// TwinCAT 3 PLC project Untitled1
// ProgramVersion: 3.1.4024.0
// libraries:
//   Tc2_MC2, * (Beckhoff Automation GmbH)
//   Tc2_Standard, * (Beckhoff Automation GmbH)
//   Tc2_System, * (Beckhoff Automation GmbH)
//   Tc2_TcpIp, * (Beckhoff Automation GmbH)
//   Tc2_Utilities, * (Beckhoff Automation GmbH)
//   Tc3_Module, * (Beckhoff Automation GmbH)
// project tree:
//   GVLs/ GVL.TcGVL, GVL_HMI.TcGVL
//   / PlcTask.TcTTO
//   POUs/Alarm/ FB_Alarm.TcPOU
//   POUs/Main/ FB_Machine.TcPOU, MAIN.TcPOU
//   POUs/UniversalBlocks/Cylinder/ FB_Cylinder.TcPOU, FB_CylinderDiag.TcPOU, FB_CylinderTemp.TcPOU, FB_CylinderTempDiag.TcPOU, FB_CylinderTempRecord.TcPOU
//   POUs/UniversalBlocks/TCP IP/ FB_TCPServer.TcPOU
//   POUs/UniversalBlocks/Universal Digital Input/ FB_Input.TcPOU, I_Input.TcIO
//   POUs/UniversalBlocks/Universal Digital Output/ FB_Output.TcPOU, I_Output.TcIO
//   POUs/UniversalBlocks/Universal motor/ FB_Axis.TcPOU, FB_Axis_Multi_Master.TcPOU, FB_HomeableAxis.TcPOU, FB_HomeableEncAxis.TcPOU, I_UniversalMotor.TcIO
// real-time tasks:
//   TASK PlcTask: cycle T#10ms, priority 20, ADS port 350
// motion (NC):
//   TASK NC-Task 1 SAF: cycle T#2ms, priority 4, ADS port 501
//   TASK NC-Task 1 SVB: cycle T#10ms, priority 8, ADS port 511
//   AXIS Axis 1 (id 1)
// variable links:
//   Untitled1 Instance <-> NC-Task 1 SAF/Axes/Axis 1
//     PlcTask Inputs/MAIN.fbMachine.servo.AxisRef.NcToPlc <-> Outputs/ToPlc
//     PlcTask Outputs/MAIN.fbMachine.servo.AxisRef.PlcToNc <-> Inputs/FromPlc

CONFIGURATION Untitled1
    RESOURCE PLC ON TwinCAT3
        TASK PlcTask(INTERVAL := T#10ms, PRIORITY := 20);
        PROGRAM MAIN WITH PlcTask : MAIN;
    END_RESOURCE
END_CONFIGURATION

// ---- GVLs/GVL.TcGVL
{attribute 'qualified_only'}
VAR_GLOBAL		
		fbLocalTime	:	FB_LocalSystemTime;
		iYear		:	UINT;
		iMonth		:	UINT;
		iDay		:	UINT;
		iHour		:	UINT;
		iMinute		:	UINT;
		iSecond		:	UINT;
END_VAR

// ---- GVLs/GVL_HMI.TcGVL
{attribute 'qualified_only'}
VAR_GLOBAL
//Cylinder
//Input
	bMoveWorkCylinder1	: BOOL;
	bMoveBaseCylinder1	: BOOL;
	bMoveWorkCylinder2	: BOOL;
	bMoveBaseCylinder2	: BOOL;
	bMoveWorkCylinder3	: BOOL;
	bMoveBaseCylinder3	: BOOL;
	bMoveWorkCylinder4	: BOOL;
	bMoveBaseCylinder4	: BOOL;
//Cylinder
//Output
	bAtBasePosCylinder1	: BOOL;
	bAtWorkPosCylinder1	: BOOL;
	bAtBasePosCylinder2	: BOOL;
	bAtWorkPosCylinder2	: BOOL;
	bAtBasePosCylinder3	: BOOL;
	bAtWorkPosCylinder3	: BOOL;
	bAtBasePosCylinder4	: BOOL;
	bAtWorkPosCylinder4	: BOOL;

//Servo
//Input
	bMoveServo			: BOOL;
	rDistance			: LREAL;
	bStopServo			: BOOL;
	
//Servo
//Output
	rPosition			: LREAL;
	rVelocity			: LREAL;
	rEnable				: BOOL;
	bErrorServo			: BOOL;
//Tcp-ip server
//Input
	bConnect			: BOOL;
	bDisconnect			: BOOL;
	bSend				: BOOL;
	sDataSend			: STRING(255);
//Tcp-ip server
//Output
	bIsConnect			: BOOL;
	sLocalHost			: T_IPv4Addr;
	sLocalPort			: UDINT;
	sDataRev			: STRING(255);
	bErrorTcp			: BOOL;
//System
//Input
	bManual				: BOOL;
	bAuto				: BOOL;
	bStart				: BOOL;
	bReset				: BOOL;
	bStopSystem			: BOOL;
	bEStopSystem		: BOOL;
	
	bSensorCheck		: BOOL;
	bSensorOK			: BOOL;
	bSensorNG			: BOOL;
	
	bSensorBase1HMI		: BOOL;
	bSensorWork1HMI     : bool;
	bSensorBase2HMI     : bool;
	bSensorWork2HMI     : bool;
	bSensorBase3HMI     : bool;
	bSensorWork3HMI     : bool;
	bSensorBase4HMI     : bool;
	bSensorWork4HMI     : bool;
	
	bRunStep			: BOOL;
	bRun				: BOOL;
	
	bOnLightGreen		: BOOL;
	bOnLightYellow		: BOOL;
	bOnLightRed			: BOOL;
		
//System
//Output
	bIsReady			: BOOL;
	bLightGreen			: BOOL;
    bLightYellow	    : bool;
    bLightRed		    : bool;
                       
	iCounterOK			: INT;
	iCounterNG			: INT;
	bErrorSystem		: BOOL;
END_VAR

// ---- POUs/UniversalBlocks/Universal Digital Input/I_Input.TcIO
INTERFACE I_Input

PROPERTY Description : STRING
GET
END_GET
SET
END_SET
END_PROPERTY

PROPERTY Value : BOOL
GET
END_GET
END_PROPERTY

END_INTERFACE

// ---- POUs/UniversalBlocks/Universal Digital Output/I_Output.TcIO
INTERFACE I_Output

PROPERTY Description : STRING
GET
END_GET
SET
END_SET
END_PROPERTY

PROPERTY ManualMode : BOOL
GET
END_GET
SET
END_SET
END_PROPERTY

PROPERTY OutAuto : BOOL
GET
END_GET
SET
END_SET
END_PROPERTY

PROPERTY OutManual : BOOL
GET
END_GET
SET
END_SET
END_PROPERTY

END_INTERFACE

// ---- POUs/UniversalBlocks/Universal motor/I_UniversalMotor.TcIO
INTERFACE I_UniversalMotor

METHOD Abort : BOOL
VAR_INPUT
END_VAR
END_METHOD

PROPERTY ActualPosition : LREAL
GET
END_GET
END_PROPERTY

PROPERTY AxisReference : AXIS_REF
GET
END_GET
END_PROPERTY

METHOD Couple : BOOL
VAR_INPUT

END_VAR

VAR

END_VAR
END_METHOD

PROPERTY Coupleable : BOOL
GET
END_GET
SET
END_SET
END_PROPERTY

PROPERTY Coupled : BOOL
GET
END_GET
END_PROPERTY

METHOD Decouple : BOOL
VAR_INPUT
END_VAR
VAR
END_VAR
END_METHOD

METHOD Home : BOOL // Start axis homing
VAR_INPUT
END_VAR
END_METHOD

PROPERTY Homed : BOOL
GET
END_GET
END_PROPERTY

PROPERTY Homingable : BOOL
GET
END_GET
SET
END_SET
END_PROPERTY

METHOD Init : BOOL
VAR_INPUT
END_VAR
END_METHOD

PROPERTY Initialized : BOOL
GET
END_GET
END_PROPERTY

METHOD Jog : BOOL
VAR_INPUT
	Distance	:	LREAL;
END_VAR
END_METHOD

PROPERTY MotorName : STRING
GET
END_GET
SET
END_SET
END_PROPERTY

METHOD MoveAbsolute : BOOL // Do action 2 request, for instance: 'Pick and place unit' change tool (additional inputs needed)
VAR_INPUT
	Position : LREAL;
END_VAR
END_METHOD

METHOD Reset : BOOL
VAR_INPUT
END_VAR
END_METHOD

PROPERTY Unit : STRING
GET
END_GET
SET
END_SET
END_PROPERTY

END_INTERFACE

// ---- POUs/Main/MAIN.TcPOU
PROGRAM MAIN
VAR
	fbMachine	: FB_Machine;
	bTimeValid	: BOOL;

END_VAR

fbMachine();
CurrentTime();

METHOD CurrentTime : BOOL
VAR_INPUT
END_VAR
GVL.fbLocalTime(bEnable := TRUE);

IF GVL.fbLocalTime.bValid THEN
	bTimeValid := TRUE;
END_IF

IF bTimeValid THEN
	GVL.iYear 	:= WORD_TO_UINT(GVL.fbLocalTime.systemTime.wYear);
	GVL.iMonth 	:= WORD_TO_UINT(GVL.fbLocalTime.systemTime.wMonth);
	GVL.iDay 	:= WORD_TO_UINT(GVL.fbLocalTime.systemTime.wDay);
	GVL.iHour 	:= WORD_TO_UINT(GVL.fbLocalTime.systemTime.wHour);
	GVL.iMinute := WORD_TO_UINT(GVL.fbLocalTime.systemTime.wMinute);
	GVL.iSecond := WORD_TO_UINT(GVL.fbLocalTime.systemTime.wSecond);
END_IF
END_METHOD

END_PROGRAM

// ---- POUs/Main/FB_Machine.TcPOU
FUNCTION_BLOCK FB_Machine
VAR_INPUT
	bManual	: FB_Input;
	bAuto	: FB_Input;
END_VAR
VAR_OUTPUT
	bError		: BOOL;
	iErrorId	: INT;
END_VAR

VAR
	iStepGeneral	: INT;
	bISError		: BOOL;
	bIsReady		: BOOL;
	trig3s			: ton :=(pt:=T#3S);
	trig1s			: ton :=(pt:=T#1S);
	trig500ms		: ton :=(pt:=T#500MS);
	trigCylin1		: ton;
	tTimeCylin1		: TIME	:= T#0.5S;
	trigCylin2		: ton;
	tTimeCylin2		: TIME	:= T#2S;
	bLightGreen		: FB_Output;
	bLightYellow	: FB_Output;
	bLightRed		: FB_Output;
	bStart			: FB_Input;
	bReset			: FB_Input;
	bSensorCheck	: FB_Input;
	bSensorOK		: FB_Input;
	bSensorNG		: FB_Input;
	bStop			: FB_Input;
	bEStop			: FB_Input;
	bStopTem		: BOOL;
	bRunStep		: BOOL := FALSE;
	bRun			: BOOL := FALSE;
	trigStep		: r_trig;
	trigSensorOK	: r_trig;
	trigSensorNG	: r_trig;
	iCounterOK		: INT;
	iCounterNG		: INT;
	bOnLightGreen	: BOOL;
	bOnLightYellow	: BOOL;
	bOnLightRed		: BOOL;
	//Tcp-ip
	trigTCp			: r_trig;
	fbTcpServer		: FB_TCPServer;
	sLocalHost		: T_IPv4Addr := '';
	nLocalPort		: UDINT := 9000;
	sNetId			: T_AmsNetId := '';  //'5.30.162.44.1.1';
	sDataRev		: STRING(255);
	sDataSend		: STRING(255);
	bConnect		: BOOL;
	bDisconnect		: BOOL;
	bSend			: BOOL;
	//servo
	servo			: FB_Axis;
	bMoveServo		: BOOL;
	rDistance		: LREAL;
	bStopServo		: BOOL;
	//cylinder
	cylinder1		: FB_CylinderDiag;
	cylinder2		: FB_CylinderDiag;
	cylinder3		: FB_CylinderDiag;
	cylinder4		: FB_CylinderDiag;
	//Alarm
	servoAlarm		: FB_Alarm;
	tcpServerAlarm	: Fb_Alarm;
	cylinderAlarm	: FB_Alarm;
	
	bMoveWorkCylinder1	: BOOL;
	bMoveBaseCylinder1	: BOOL;
	bMoveWorkCylinder2	: BOOL;
	bMoveBaseCylinder2	: BOOL;
	bMoveWorkCylinder3	: BOOL;
	bMoveBaseCylinder3	: BOOL;
	bMoveWorkCylinder4	: BOOL;
	bMoveBaseCylinder4	: BOOL;
	
	bManualHMI		: BOOL;
	bAutoHMI		: BOOL;
	bStartHMI		: BOOL;
	bResetHMI		: bool;
	bStopHMI		: bool;
	bEStopHMI		: bool;
	bSensorCheckHMI	: bool;
	bSensorOKHMI	: bool;
	bSensorNGHMI	: BOOL;
	bSensorBase1HMI	: BOOL;
	bSensorWork1HMI	: BOOL;
	bSensorBase2HMI	: BOOL;
	bSensorWork2HMI	: BOOL;
	bSensorBase3HMI	: BOOL;
	bSensorWork3HMI	: BOOL;
	bSensorBase4HMI	: BOOL;
	bSensorWork4HMI	: BOOL;
	
	iStepRun: INT := 0;
	iStepAuto: INT := 0;
	bCheck : BOOL;
	bFirstCycle	: BOOL := TRUE;
END_VAR

StateMachine();
AssignHMI();
servo();
fbTcpServer();
//Menu mode
IF bManual.Value OR bManualHMI THEN
	iStepRun	:= 20;
END_IF
IF bAuto.Value OR bAutoHMI THEN
	iStepRun	:= 10;
END_IF
//Reset
IF bReset.Value OR bResetHMI THEN
	iStepGeneral := 0;
END_IF
//Stop
IF bStop.Value OR bStopHMI THEN
	bStopTem := TRUE;
END_IF
IF bEStop.Value OR bEStopHMI THEN
	iStepGeneral	:= 99;
END_IF
//Error
bError := servoAlarm.Get() OR tcpServerAlarm.Get() OR cylinderAlarm.Get();

METHOD AssignHMI : BOOL
VAR_INPUT
END_VAR
//Cylinder              
//Input                 
bMoveWorkCylinder1		:=	GVL_HMI.bMoveWorkCylinder1	;
bMoveBaseCylinder1		:=	GVL_HMI.bMoveBaseCylinder1	;
bMoveWorkCylinder2		:=	GVL_HMI.bMoveWorkCylinder2	;
bMoveBaseCylinder2		:=	GVL_HMI.bMoveBaseCylinder2	;
bMoveWorkCylinder3		:=	GVL_HMI.bMoveWorkCylinder3	;
bMoveBaseCylinder3		:=	GVL_HMI.bMoveBaseCylinder3	;
bMoveWorkCylinder4		:=	GVL_HMI.bMoveWorkCylinder4	;
bMoveBaseCylinder4		:=	GVL_HMI.bMoveBaseCylinder4	;

bSensorBase1HMI			:= GVL_HMI.bSensorBase1HMI;
bSensorWork1HMI         := GVL_HMI.bSensorWork1HMI;
bSensorBase2HMI         := GVL_HMI.bSensorBase2HMI;
bSensorWork2HMI         := GVL_HMI.bSensorWork2HMI;
bSensorBase3HMI         := GVL_HMI.bSensorBase3HMI;
bSensorWork3HMI         := GVL_HMI.bSensorWork3HMI;
bSensorBase4HMI         := GVL_HMI.bSensorBase4HMI;
bSensorWork4HMI         := GVL_HMI.bSensorWork4HMI;
//Cylinder                                          
//Output                
GVL_HMI.bAtBasePosCylinder1	:= cylinder1.bState_AtBasePos OR cylinder1.bState_MoveToBase;
GVL_HMI.bAtWorkPosCylinder1	:= cylinder1.bState_AtWorkPos OR cylinder1.bState_MoveToWork;
GVL_HMI.bAtBasePosCylinder2	:= cylinder2.bState_AtBasePos OR cylinder2.bState_MoveToBase;
GVL_HMI.bAtWorkPosCylinder2	:= cylinder2.bState_AtWorkPos OR cylinder2.bState_MoveToWork;
GVL_HMI.bAtBasePosCylinder3	:= cylinder3.bState_AtBasePos OR cylinder3.bState_MoveToBase;
GVL_HMI.bAtWorkPosCylinder3	:= cylinder3.bState_AtWorkPos OR cylinder3.bState_MoveToWork;
GVL_HMI.bAtBasePosCylinder4	:= cylinder4.bState_AtBasePos OR cylinder4.bState_MoveToBase;
GVL_HMI.bAtWorkPosCylinder4	:= cylinder4.bState_AtWorkPos OR cylinder4.bState_MoveToWork;
                        
//Servo                 
//Input                 
bMoveServo	:=	GVL_HMI.bMoveServo	;		
rDistance	:=	GVL_HMI.rDistance	;		
bStopServo	:=	GVL_HMI.bStopServo	;		
	                    
//Servo                 
//Output                
GVL_HMI.rPosition	:= servo.ActualPosition;		
GVL_HMI.rVelocity	:= servo.ActualVelocity;
GVL_HMI.rEnable		:= servo.Enabled;	
gvl_hmi.bErrorServo	:= servo.AnyError;
//Tcp-ip server         
//Input                 
bConnect	:= GVL_HMI.bConnect		;	
bDisconnect	:= GVL_HMI.bDisconnect	;		
bSend		:= GVL_HMI.bSend		;		
sDataSend	:= GVL_HMI.sDataSend	;
fbTcpServer.LocalHost	:=GVL_HMI.sLocalHost;
fbTcpServer.LocalPort	:=GVL_HMI.sLocalPort;		
//Tcp-ip server         
//Output                
GVL_HMI.bIsConnect	:= fbTcpServer.IsConnect;		
GVL_HMI.sDataRev	:= fbTcpServer.DataRev;
GVL_HMI.bErrorTcp	:= fbTcpServer.Error;
//System                
//Input                 
bRunStep			:= gvl_hmi.bRunStep;
bRun	            := gvl_hmi.bRun;
bManualHMI			:= GVL_HMI.bManual		;		
bAutoHMI			:= GVL_HMI.bAuto		;		
bStartHMI			:= GVL_HMI.bStart		;		
bResetHMI			:= GVL_HMI.bReset		;		
bStopHMI			:= GVL_HMI.bStopSystem	;		 	
bEStopHMI			:= GVL_HMI.bEStopSystem	;		                 
bSensorCheckHMI		:= GVL_HMI.bSensorCheck	;		
bSensorOKHMI		:= GVL_HMI.bSensorOK	;		
bSensorNGHMI		:= GVL_HMI.bSensorNG	;
bOnLightGreen			:= gvl_hmi.bOnLightGreen;
bOnLightYellow		:= gvl_hmi.bOnLightGreen;
bOnLightRed		  	:= gvl_hmi.bOnLightGreen;
		                
//System                
//Output

gvl_hmi.bIsReady		:= bIsReady;               
GVL_HMI.iCounterOK		:= iCounterOK;	
GVL_HMI.iCounterNG		:= iCounterOK;		
GVL_HMI.bErrorSystem	:= bError;

GVL_HMI.bLightGreen		:= 	bLightGreen.OutAuto;
GVL_HMI.bLightYellow    :=  bLightYellow.OutAuto;
GVL_HMI.bLightRed	    :=  bLightRed.OutAuto;
END_METHOD

METHOD PRIVATE StateAuto : BOOL
VAR

END_VAR

CASE iStepAuto OF
	0: //run servo 10
			trigStep(clk:=bRun);
			IF NOT bRunStep OR trigStep.Q THEN
				iStepAuto := iStepAuto + 1;
			END_IF
	1:
		IF NOT servo.AnyError AND servo.Enabled THEN
			IF servo.ActualPosition <> 10 THEN
				servo.MoveAbsolute(Position := 10);
			END_IF
		ELSE
			iStepAuto := 99;
		END_IF
		IF servo.ActualPosition = 10 THEN
			trigStep(clk:=bRun);
			IF NOT bRunStep OR trigStep.Q THEN
				iStepAuto := iStepAuto + 1;
			END_IF
		END_IF

	2: // run cylinder 1
		IF bSensorCheck.Value OR bSensorCheckHMI THEN
			bCheck := TRUE;
		END_IF		
		
		IF bCheck THEN
			IF NOT cylinder1.bError THEN
				cylinder1.MoveToWork();
			ELSE
				iStepAuto	:= 99;
			END_IF
			trigCylin1(in:= cylinder1.bState_AtWorkPos OR bSensorWork1HMI,pt:=tTimeCylin1);
			IF trigCylin1.Q THEN
				cylinder1.MoveToBase();
				bCheck	:= FALSE;
			END_IF
		END_IF
			
			
		IF cylinder1.bState_AtBasePos OR bSensorBase1HMI AND( NOT bSensorCheck.Value OR NOT bSensorCheckHMI )THEN
			trigStep(clk:=bRun);
			IF NOT bRunStep OR trigStep.Q THEN
				iStepAuto := iStepAuto + 1;
			END_IF
		END_IF
	3:// run servo 70
		IF NOT servo.AnyError THEN
			IF servo.ActualPosition <> 70 THEN
				servo.MoveAbsolute(Position := 70);
			END_IF			
		ELSE
			iStepAuto := 99;
		END_IF
		IF servo.ActualPosition = 70 THEN
			bCheck	:= TRUE;
			trigStep(clk:=bRun);
			IF NOT bRunStep OR trigStep.Q THEN
				iStepAuto := iStepAuto + 1;
			END_IF
		END_IF
		
	4://run cylin 2
		IF bCheck THEN
			IF NOT cylinder2.bError THEN
				cylinder2.MoveToWork();
			ELSE
				iStepAuto	:= 99;
			END_IF
			trigCylin2(in:= cylinder2.bState_AtWorkPos OR bSensorWork2HMI,pt:=tTimeCylin2);
			IF trigCylin2.Q THEN
				cylinder2.MoveToBase();
				bCheck	:= FALSE;
			END_IF
		END_IF
		IF NOT bCheck THEN
			trigStep(clk:=bRun);
			IF NOT bRunStep OR trigStep.Q THEN
				iStepAuto := iStepAuto + 1;
			END_IF
		END_IF

	5://run servo 130
		IF NOT servo.AnyError THEN
			IF servo.ActualPosition <> 130 THEN
				servo.MoveAbsolute(Position := 130);
			END_IF
		ELSE
			iStepAuto := 99;
		END_IF
		
		IF servo.ActualPosition = 130 THEN
			bCheck	:= TRUE;
			trigStep(clk:=bRun);
			IF NOT bRunStep OR trigStep.Q THEN
				iStepAuto := iStepAuto + 1;
			END_IF
		END_IF
	6:// trigger camera
		IF bCheck THEN
			IF fbTcpServer.IsConnect THEN
				fbTcpServer.SendData(DataSend :='CHE,1');
				bCheck := FALSE;
			ELSE
				iStepAuto := 99;
			END_IF
		END_IF
	
		IF NOT bCheck THEN
			trigStep(clk:=bRun);
			IF NOT bRunStep OR trigStep.Q THEN
				iStepAuto := iStepAuto + 1;
			END_IF
		END_IF
	
	7:// check camera
		sDataRev := fbTcpServer.DataRev;
		trigStep(clk:=bRun);
		IF NOT bRunStep OR trigStep.Q THEN
			IF sDataRev = 'CAM,1,OK' THEN
					iStepAuto := iStepAuto + 1;
			END_IF
			IF sDataRev = 'CAM,1,NG' THEN
					iStepAuto := iStepAuto + 2;
			END_IF
		END_IF
		
	8:// run servo 190
		IF NOT servo.AnyError THEN
			IF servo.ActualPosition <> 190 THEN
				servo.MoveAbsolute(Position := 190);
			END_IF
		ELSE
			iStepAuto := 99;
		END_IF
		
		IF servo.ActualPosition = 190 THEN
			bCheck	:= TRUE;
			trigStep(clk:=bRun);
			IF NOT bRunStep OR trigStep.Q THEN
				iStepAuto := iStepAuto + 2;
			END_IF
		END_IF

	9:// run servo 210
		IF NOT servo.AnyError THEN
			IF servo.ActualPosition <> 210 THEN
				servo.MoveAbsolute(Position := 210);
			END_IF
		ELSE
			iStepAuto := 99;
		END_IF
		IF servo.ActualPosition = 210 THEN
			bCheck	:= TRUE;
			trigStep(clk:=bRun);
			IF NOT bRunStep OR trigStep.Q THEN
				iStepAuto := iStepAuto + 2;
			END_IF
		END_IF
	10://run cylin 3
		IF bCheck THEN
			IF NOT cylinder3.bError THEN
				cylinder3.MoveToWork();
				IF cylinder3.bState_AtWorkPos OR bSensorWork3HMI THEN
					cylinder3.MoveToBase();
					bCheck := FALSE;
				END_IF
			ELSE
				iStepAuto	:= 99;
			END_IF
		END_IF
		
		IF NOT bCheck THEN
			trigStep(clk:=bRun);
			IF NOT bRunStep OR trigStep.Q THEN
				iStepAuto := iStepAuto + 2;
			END_IF
		END_IF

	11://run cylin 4
		IF bCheck THEN
			IF NOT cylinder4.bError THEN
				cylinder4.MoveToWork();
				IF cylinder4.bState_AtWorkPos OR bSensorWork4HMI THEN
					cylinder4.MoveToBase();
					bCheck := FALSE;
				END_IF
			ELSE
				iStepAuto	:= 99;
			END_IF
		END_IF
		
		IF NOT bCheck THEN
			trigStep(clk:=bRun);
			IF NOT bRunStep OR trigStep.Q THEN
				iStepAuto := iStepAuto + 1;
			END_IF
		END_IF

	12:// counter
		trigSensorOK(clk:=bSensorOK.Value OR bSensorOKHMI);
		trigSensorNG(clk:=bSensorNG.Value OR bSensorNGHMI);
		IF trigSensorOK.Q THEN
			icounterOK := icounterOK + 1;
		END_IF
		IF trigSensorNG.Q THEN
			icounterNG := icounterNG + 1;
		END_IF
		IF NOT bStopTem THEN
			iStepAuto := 0;
		END_IF
	99://Error
		iStepGeneral := 99;
		
		
END_CASE
END_METHOD

METHOD PRIVATE StateError : BOOL
VAR
	bfirstCycle	: bool := true;
END_VAR
IF bfirstCycle THEN
	bfirstCycle:= FALSE;
	IF servo.AnyError THEN
		servoAlarm.Set(bIn := TRUE);
		servoAlarm.Description := 'Servo bi loi';
	END_IF
	IF fbTcpServer.Error THEN
		tcpServerAlarm.Set(bIn := TRUE);
		tcpServerAlarm.Description := 'TCP-IP Server bi loi';
		END_IF
	IF NOT fbTcpServer.IsConnect THEN
		tcpServerAlarm.Set(bIn := TRUE);
		tcpServerAlarm.Description := 'Khong co Client nao ket noi';
	END_IF
END_IF
	

trig1s(IN := TRUE);
IF trig1s.Q THEN
	trig1s(IN := TRUE);
	bLightRed.OutAuto := NOT bLightRed.OutAuto;
END_IF

IF bReset.Value THEN
	iStepGeneral := 0;
END_IF
END_METHOD

METHOD PRIVATE StateInit : BOOL
VAR
	
END_VAR
//init cylin
cylinder1.MoveToBase();
cylinder1.Reset();
cylinder2.MoveToBase();
cylinder2.Reset();
cylinder3.MoveToBase();
cylinder3.Reset();
cylinder4.MoveToBase();
cylinder4.Reset();
//init servo
servo.Reset();
servo.Override := 100;
servo.Init();
servo.MoveAbsolute(Position:=0);
//Init tcp-ip
IF NOT fbTcpServer.IsConnect THEN
	IF bFirstCycle THEN
		bFirstCycle := FALSE;
		fbTcpServer.Disconnect();
		fbTcpServer.LocalHost	:= sLocalHost;
		fbTcpServer.LocalPort	:= nLocalPort;
		fbTcpServer.NetId		:= sNetId;
		fbTcpServer.Connect();
	END_IF
END_IF

bLightGreen.OutAuto 	:= FALSE;
bLightYellow.OutAuto 	:= FALSE;
blightRed.OutAuto 		:= FALSE;

bCheck					:= FALSE;
iStepAuto				:= 0;
IF servo.ActualPosition = 0 THEN
	iStepGeneral			:= iStepGeneral + 1;
END_IF
END_METHOD

METHOD private StateMachine : BOOL
VAR_INPUT
END_VAR
CASE iStepGeneral OF
	0: 
		StateInit();
	1:
		StateUninitialized();
	2:
		StateReady();
	10:
		StateRun();
	20:
		StateRunDone();
	30:
		StateStop();
	40:
		StateStopDone();
	99:
		StateError();
	
END_CASE
END_METHOD

METHOD PRIVATE StateManual : BOOL
VAR_INPUT
END_VAR
//cylinder
IF bMoveWorkCylinder1 THEN
	cylinder1.MoveToWork();
	bMoveWorkCylinder1 := FALSE;
END_IF
IF bMoveBaseCylinder1 THEN
	cylinder1.MoveToBase();
	bMoveBaseCylinder1 := FALSE;
END_IF
IF bMoveWorkCylinder2 THEN
	cylinder2.MoveToWork();
	bMoveWorkCylinder2 := FALSE;
END_IF
IF bMoveBaseCylinder2 THEN
	cylinder2.MoveToBase();
	bMoveBaseCylinder2 := FALSE;
END_IF
IF bMoveWorkCylinder3 THEN
	cylinder3.MoveToWork();
	bMoveWorkCylinder3 := FALSE;
END_IF
IF bMoveBaseCylinder3 THEN
	cylinder3.MoveToBase();
	bMoveBaseCylinder3 := FALSE;
END_IF
IF bMoveWorkCylinder4 THEN
	cylinder4.MoveToWork();
	bMoveWorkCylinder4 := FALSE;
END_IF
IF bMoveBaseCylinder4 THEN
	cylinder4.MoveToBase();
	bMoveBaseCylinder4 := FALSE;
END_IF
//servo
IF bMoveServo THEN
	servo.Jog(Distance:=rDistance);
	bMoveServo := FALSE;
END_IF
IF bStopServo THEN
	bStopServo := FALSE;
	servo.Stop();
END_IF
//TCP-Ip
IF bConnect THEN
	fbTcpServer.Connect();
	bConnect := FALSE;
END_IF
IF bDisconnect THEN
	fbTcpServer.Disconnect();
	bDisconnect := FALSE;
END_IF
IF bSend THEN
	fbTcpServer.SendData(DataSend := sDataSend);
	bSend := FALSE;
END_IF
//system
bLightGreen.OutAuto		:= bOnLightGreen	;
bLightYellow.OutAuto    := bOnLightYellow	;
bLightRed.OutAuto       := bOnLightRed		;
END_METHOD

METHOD PRIVATE StateReady : BOOL
VAR_INPUT
END_VAR
trig500ms(in := TRUE);
IF bIsReady AND trig500ms.Q THEN
	trig500ms(in := FALSE);
	bLightGreen.OutAuto := NOT bLightGreen.OutAuto;
END_IF

IF bStart.Value OR bStartHMI THEN
	iStepGeneral := 10;
END_IF
END_METHOD

METHOD PRIVATE StateRun : BOOL
VAR_INPUT
END_VAR
CASE iStepRun OF
	10:
		StateAuto();
		bLightGreen.OutAuto := TRUE;
	20:
		StateManual();
END_CASE
END_METHOD

METHOD PRIVATE StateRunDone : BOOL
VAR_INPUT
END_VAR
END_METHOD

METHOD PRIVATE StateStop : BOOL
VAR_INPUT
END_VAR
END_METHOD

METHOD PRIVATE StateStopDone : BOOL
VAR_INPUT
END_VAR
END_METHOD

METHOD PRIVATE StateUninitialized : BOOL
VAR_INPUT
END_VAR
bISError := servo.AnyError OR fbTcpServer.Error OR fbTcpServer.Error ;
//bIsReady := cylinder1.bState_AtBasePos AND cylinder2.bState_AtBasePos AND cylinder3.bState_AtBasePos AND cylinder4.bState_AtBasePos AND fbTcpServer.IsConnect AND servo.Enabled;
bIsReady := TRUE;
		
IF bIsError THEN
	iStepGeneral := 99;
END_IF

IF NOT bIsReady THEN
	bLightYellow.OutAuto := TRUE;
END_IF

IF bIsReady THEN
	iStepGeneral := 2;
END_IF
IF NOT bIsReady THEN
	IF bReset.Value OR bResetHMI THEN
		iStepGeneral := 0;
	END_IF
END_IF
END_METHOD

END_FUNCTION_BLOCK

// ---- POUs/UniversalBlocks/Universal Digital Input/FB_Input.TcPOU
FUNCTION_BLOCK FB_Input IMPLEMENTS I_Input
VAR_INPUT
END_VAR
VAR_OUTPUT
END_VAR
VAR
	sDescription			:	STRING; //Description of the physical input
	bIn				AT %I*	:	BOOL;	// Physical input
	bRisingTrigger			:	BOOL;
	bFallingTrigger			:	BOOL;
	rtIn					:	R_TRIG; //Rising edge of the input
	ftIn					:	F_TRIG; //Falling edge of the input	
END_VAR

PROPERTY Description : STRING
GET
Description := sDescription;
END_GET
SET
sDescription := Description;
END_SET
END_PROPERTY

PROPERTY Value : BOOL
GET
Value := bIn;
END_GET
END_PROPERTY

END_FUNCTION_BLOCK

// ---- POUs/UniversalBlocks/Universal Digital Output/FB_Output.TcPOU
// Function block used for physical output control
FUNCTION_BLOCK FB_Output IMPLEMENTS I_Output
VAR_INPUT

END_VAR
VAR_OUTPUT

END_VAR
VAR
	bOut	AT %Q*	:	BOOL;	// Physical output
	sDescription	:	STRING;	// Description of the output
	bOutAuto		:	BOOL;	// This value will be used in automatic mode
	bManualMode		:	BOOL;	// Turns on and off manual mode
	bOutManual		:	BOOL;	// This value will be used in manual mode
END_VAR

{attribute 'monitoring' := 'variable'}
PROPERTY Description : STRING
GET
Description := sDescription;
END_GET
SET
sDescription := Description;
END_SET
END_PROPERTY

{attribute 'monitoring' := 'variable'}
PROPERTY ManualMode : BOOL
GET
ManualMode := bManualMode;
END_GET
SET
bManualMode := ManualMode;
END_SET
END_PROPERTY

{attribute 'monitoring' := 'variable'}
PROPERTY OutAuto : BOOL
GET
OutAuto := bOut;
END_GET
SET
bOutAuto := OutAuto;
IF NOT bManualMode THEN
	bOut := bOutAuto;
END_IF
END_SET
END_PROPERTY

{attribute 'monitoring' := 'variable'}
PROPERTY OutManual : BOOL
GET
OutManual := bOut;
END_GET
SET
bOutManual := OutManual;
IF bManualMode THEN
	bOut := bOutManual;
END_IF
END_SET
END_PROPERTY

END_FUNCTION_BLOCK

// ---- POUs/UniversalBlocks/TCP IP/FB_TCPServer.TcPOU
FUNCTION_BLOCK FB_TCPServer

VAR
	sLocalHost: T_IPv4Addr;
	nLocalPort: UDINT := 9000;
	//bStartCommunication : BOOL;
	sNetId	:T_AmsNetId;
	//bSent	: BOOL;

	bConnected: BOOL;
	sSendData: STRING(255);
	bBusy: BOOL;	
	bError: BOOL;
	nErrorID: UDINT;
	sDataRev: STRING(255);

	//iState: INT;
	hListener: T_HSOCKET;
	hSocket: T_HSOCKET;
	fbSocketAccept: FB_SocketAccept;
	fbSocketListen: FB_SocketListen;
	fbSocketReceive: FB_SocketReceive;
	fbSocketClose: FB_SocketClose;
	fbSocketCloseAll: FB_SocketCloseAll;
	fbSocketSend: FB_SocketSend;
	bAcceptExecute: BOOL;
	sReadData: STRING(255);
	ReceiveCounter: UDINT;
	bSocketCloseError: BOOL;
	nSocketCloseError: UDINT;
	//bSendTrigger: BOOL;
	//sData : STRING(255);
	iStepGeneral	: INT := 0;
	iStepStop		: INT := 0;
END_VAR

StateMachine();
IF bError THEN
	iStepGeneral := 50;
END_IF

METHOD Connect : BOOL
VAR_INPUT
END_VAR
IF NOT bConnected AND NOT bError THEN
	iStepGeneral := 1;
END_IF
END_METHOD

PROPERTY DataRev : String(255)
GET
DataRev := sDataRev;
END_GET
END_PROPERTY

METHOD Disconnect : BOOL
VAR_INPUT
END_VAR
iStepGeneral := 50;
END_METHOD

PROPERTY Error : bool
GET
Error	:= bError;
END_GET
END_PROPERTY

PROPERTY IsConnect : bool
GET
IsConnect	:= bConnected;
END_GET
END_PROPERTY

PROPERTY LocalHost : T_IPv4Addr
SET
sLocalHost	:= LocalHost;
END_SET
END_PROPERTY

PROPERTY LocalPort : UDINT
SET
//nLocalPort	:= LocalPort;
END_SET
END_PROPERTY

PROPERTY NetId : T_AmsNetId
SET
sNetId	:= NetId;
END_SET
END_PROPERTY

METHOD SendData : BOOL
VAR_INPUT
	DataSend	: STRING(255);
END_VAR
sSendData := DataSend;
IF bConnected OR bError THEN
	IF iStepGeneral = 30 THEN
		iStepGeneral := 40;
	END_IF
END_IF
END_METHOD

METHOD private StateAccept : BOOL
VAR_INPUT
END_VAR
fbSocketAccept(																
		sSrvNetId:= sNetId, 		
		hListener:= hListener, 													
		bExecute:= TRUE, 
		tTimeout:= T#4S, 
		bAccepted=> , 
		bBusy=> bBusy, 
		bError=> bError, 
		nErrId=> nErrorID,
		hSocket=> hSocket);														
	IF NOT fbSocketAccept.bBusy THEN
		fbSocketAccept(bExecute:= FALSE);
	END_IF

	IF bError THEN
		iStepGeneral := 50; 
	ELSIF hSocket.handle <> 0 THEN
		iStepGeneral := iStepGeneral + 10; 
		bConnected := TRUE;
	END_IF
END_METHOD

METHOD PRIVATE StateClose : BOOL
VAR_INPUT
END_VAR
CASE iStepStop OF
0:	// Error Handling	
	fbSocketClose(																// Close Listener-Socket
		sSrvNetId:= sNetId, 
		hSocket:= hListener, 
		bExecute:= TRUE, 
		tTimeout:= T#4S, 
		bBusy=> , 
		bError=> bError, 
		nErrId=> nErrorID);		
	IF (NOT fbSocketClose.bBusy) OR fbSocketClose.bError THEN
		hListener.handle := 0;
		iStepStop := iStepStop + 1;
	END_IF
1:	
	fbSocketClose(bExecute := FALSE);
	iStepStop := iStepStop + 1;
2:
	fbSocketClose(																// Close Connection Socket
		sSrvNetId:= sNetId, 
		hSocket:= hSocket, 
		bExecute:= TRUE, 
		tTimeout:= T#4S, 
		bBusy=> , 
		bError=> bError, 
		nErrId=> nErrorID);
	IF NOT (fbSocketClose.bBusy) OR fbSocketClose.bError THEN
		hSocket.handle 	:= 0;	
		iStepGeneral 	:= 0;
		iStepStop		:= 0;
		bConnected 		:= FALSE;
	END_IF
END_CASE
END_METHOD

METHOD PRIVATE StateInit : BOOL
VAR_INPUT
END_VAR
fbSocketCloseAll(
		sSrvNetId:= sNetId, 
		bExecute:= TRUE, 
		tTimeout:= T#3S, 
		bBusy=> , 
		bError=> bSocketCloseError, 
		nErrId=> nSocketCloseError);

IF NOT (fbSocketCloseAll.bBusy OR fbSocketCloseAll.bError) THEN
		fbSocketCloseAll(bExecute:= FALSE);
		fbSocketListen(bExecute := FALSE);
		fbSocketAccept(bExecute := FALSE);
		fbSocketClose(bExecute:= FALSE);
		bConnected	:= FALSE;
		bBusy 		:= TRUE;
		iStepGeneral := 10;
END_IF
END_METHOD

METHOD PRIVATE StateListen : BOOL
VAR_INPUT
END_VAR
fbSocketListen(																
		sSrvNetId:= sNetId, 														
		sLocalHost:= sLocalHost, 												
		nLocalPort:= nLocalPort, 												
		bExecute:= TRUE, 
		tTimeout:= T#4S, 
		bBusy=> bBusy, 
		bError=> bError, 
		nErrId=> nErrorID,
		hListener=> hListener);													
		
	IF hListener.handle <> 0 THEN
		iStepGeneral := iStepGeneral + 10;	
	ELSIF bError THEN
		iStepGeneral := 50;
	END_IF
END_METHOD

METHOD PRIVATE StateMachine : BOOL
VAR_INPUT
END_VAR
CASE iStepGeneral OF
	1:
		StateInit();
	10:
		StateListen();
	20:
		StateAccept();
	30:
		StateReceive();
	40:
		StateSend();
	50:
		StateClose();
END_CASE
END_METHOD

METHOD PRIVATE StateReceive : BOOL
VAR_INPUT
END_VAR
fbSocketReceive(															
		sSrvNetId:= sNetId, 
		hSocket:= hSocket, 
		cbLen:= SIZEOF(sReadData) , 
		pDest:= ADR(sReadData), 
		bExecute:= TRUE, 														
		tTimeout:= T#4S, 
		bBusy=> , 
		bError=> bError, 
		nErrId=> nErrorID,
		nRecBytes=> );
		
	IF NOT fbSocketReceive.bBusy THEN
		fbSocketReceive(bExecute := FALSE);
		IF fbSocketReceive.nRecBytes <> 0 THEN									
			sDataRev := sReadData;
		END_IF
	END_IF
	
	IF fbSocketReceive.bError OR(NOT bConnected) THEN					
		iStepGeneral := 50;
	END_IF
END_METHOD

METHOD PRIVATE StateSend : BOOL
VAR_INPUT
END_VAR
fbSocketSend(																// Send Data to client
		sSrvNetId:= sNetId, 
		hSocket:= hSocket, 
		cbLen:= SIZEOF(sSendData), 
		pSrc:= ADR(sSendData),
		bExecute:= TRUE, 
		tTimeout:= T#3S, 
		bBusy=> , 
		bError=> bError, 
		nErrId=> nErrorID);	
	
	IF NOT fbSocketSend.bBusy THEN												// Switch back to receiving state after sending
		iStepGeneral := iStepGeneral - 10;
	ELSIF fbSocketSend.bError OR NOT bConnected THEN
		iStepGeneral := 50;													// Close connection in case of error 
	END_IF
END_METHOD

END_FUNCTION_BLOCK

// ---- POUs/UniversalBlocks/Universal motor/FB_Axis.TcPOU
FUNCTION_BLOCK FB_Axis IMPLEMENTS I_UniversalMotor
VAR_OUTPUT

END_VAR
VAR	
		// =============== Axis reference =========================
	AxisRef			: AXIS_REF;				// Axis reference (process data plc/nc)
	
	//Motors data
	sMotorName	:	STRING := 'Motor';
	sUnits		:	STRING := 'mm';


	iNumberOfInstance	: SINT := 1; //numebr of currently used instance of MC_MoveVelocity
	// =============== Done signals of Halt and Reset =========
	bResetDone		: BOOL;					// Status of function block MC_Reset
	bHaltDone		: BOOL;					// Status of function block MC_Halt

	// =============== State variables ========================
	bStatusEnable	: BOOL;					// Enable feedback
	
	// =============== Motion parameters, override =====================
	lrVelocityAuto			: LREAL := 2;			// Target velocity
	lrAccelerationAuto		: LREAL := 100;			// Target acceleration
	lrDecelerationAuto		: LREAL := 100;			// Target deceleration
	lrJerkAuto				: LREAL := 100;			// Target jerk
	lrVelocityManual		: LREAL := 2;			// Target velocity
	lrAccelerationManual	: LREAL := 100;			// Target acceleration
	lrDecelerationManual	: LREAL := 100;			// Target deceleration
	lrJerkManual			: LREAL := 100;			// Target jerk
	lrOverride 				: LREAL := 100.0;		// Override 100%
	lrPosition				: LREAL := 0;			// Target Position
	mcBufferMode			: MC_BufferMode := MC_Aborting;		// buffer mode standard value
	lrDistanceToGo			: LREAL := 0; 			// distance do go for relative movement
	lrActualPosition		: LREAL; // actual postion
	
	// =============== Trigger function blocks ================
	fbTriggerHalt	: R_TRIG;				// Trigger to recognize rising edge of halt input
	fbTriggerReset	: R_TRIG;				// Trigger to recognize rising edge of reset input
	
//	// =============== Axis reference =========================
//	AxisRef			: AXIS_REF;				// Axis reference (process data plc/nc)
	
	// =============== Motion function blocks =================
	fbMcPower 		: MC_Power;				// FB for enable and override
	fbMcReset 		: MC_Reset;				// FB to reset axis
	fbMcStop 		: MC_Stop;				// FB to stop axis
	fbMcHalt		: MC_Halt;				// FB to halt axis

	fbMcMoveVelocity		: MC_MoveVelocity;		// FB to move axis (velocity movement)
	fbMcMoveAbsolute		: MC_MoveAbsolute;		// FB to move axis (absolute PTP movement)
	fbMcMoveRelative		: MC_MoveRelative;		// FB to move axis (relative PTP movement)
	fbReadActualVelocity	: MC_ReadActualVelocity; //FB to read actual velocity of axis
	fbReadActualPosition	: MC_ReadActualPosition;//FB to read actual position of axis
	
	bFirstCycle		:	BOOL := TRUE; // indicates first cycle
	iStepInit		:	INT; // step of initialization
	

	bMoveVelocity	:	BOOL; //do action 2 variable
	bMoveAbsolute	:	BOOL; //do action 3 variable
	bMoveRelative	:	BOOL; //do action 4 variable
	bStop			:	BOOL; //do action 5 variable

	iStepGeneral	:	INT; // step of main state of unit
	iStepAborting	:	INT;

	
	bManualMode		:	BOOL;
	
	
	fbAxisError		:	FB_Alarm;
	
	bCoupleable		:	BOOL;
	bHomingable		:	BOOL;
	bInitialized	:	BOOL;

	// =============== Error variables ========================
	bError			: BOOL;					// Error signal
	iErrorID		: UDINT;				// Error ID
	
END_VAR

IF bFirstCycle THEN
	bFirstCycle := FALSE;
END_IF
// cyclic
		StateMachine();
		
	// reset commands
		bMoveVelocity := FALSE;
		bMoveAbsolute := FALSE;
		bMoveRelative := FALSE;
		bStop := FALSE;
		
	// read error
		IF AxisRef.Status.Error THEN
			bError := TRUE;
			iErrorID :=  AxisRef.Status.ErrorID;
		END_IF
		
	// read pos
		fbReadActualPosition(Enable := TRUE, Axis:=AxisRef);
		lrActualPosition :=	fbReadActualPosition.Position;

	// error	
		//fbAxisError.Description := FUN_MergeStrings5(sMotorName, ' axis error number: ', UDINT_TO_STRING(iErrorID), '', '');
		//fbAxisError.Set(bError);

	// status bits
		bInitialized := iStepGeneral > 10;

METHOD Abort : BOOL // Abort axis, it will disable the power
VAR_INPUT
END_VAR
IF iStepGeneral <> 0 THEN
	iStepGeneral := -10;
END_IF
iStepInit := 0;

//Method output
	Abort := (iStepGeneral = 0);
END_METHOD

{attribute 'monitoring' := 'variable'}
PROPERTY AccelerationAuto : LREAL
GET
AccelerationAuto := lrAccelerationAuto;
END_GET
SET
lrAccelerationAuto := AccelerationAuto;
END_SET
END_PROPERTY

{attribute 'monitoring' := 'variable'}
PROPERTY AccelerationManual : LREAL
GET
AccelerationManual := lrAccelerationManual;
END_GET
SET
lrAccelerationManual := AccelerationManual;
END_SET
END_PROPERTY

{attribute 'monitoring' := 'variable'}
PROPERTY ActualPosition : LREAL
GET
ActualPosition := lrActualPosition;
END_GET
END_PROPERTY

{attribute 'monitoring' := 'variable'}
PROPERTY ActualVelocity : LREAL
GET
fbReadActualVelocity(Enable:=TRUE,Axis:=AxisRef);
ActualVelocity:=fbReadActualVelocity.ActualVelocity;
END_GET
END_PROPERTY

{attribute 'monitoring' := 'variable'}
PROPERTY AnyError : BOOL
GET
AnyError := bError;
END_GET
END_PROPERTY

PROPERTY AxisReference : AXIS_REF
GET
AxisReference := AxisRef;
END_GET
END_PROPERTY

{attribute 'monitoring' := 'variable'}
PROPERTY Buffering : BOOL // TRUE for Enable, FALSE for disable
SET
IF Buffering THEN
	mcBufferMode := MC_BlendingNext;
ELSE
	mcBufferMode := MC_Aborting;
END_IF;
END_SET
END_PROPERTY

METHOD Couple : BOOL
VAR_INPUT
END_VAR
VAR
END_VAR
END_METHOD

{attribute 'monitoring' := 'variable'}
PROPERTY Coupleable : BOOL
GET
Coupleable := bCoupleable;
END_GET
SET
bCoupleable := Coupleable;
END_SET
END_PROPERTY

{attribute 'monitoring' := 'variable'}
PROPERTY Coupled : BOOL
GET
Coupled := AxisRef.Status.Coupled;
END_GET
END_PROPERTY

{attribute 'monitoring' := 'variable'}
PROPERTY DecelerationAuto : LREAL
GET
DecelerationAuto := lrDecelerationAuto;
END_GET
SET
lrDecelerationAuto := DecelerationAuto;
END_SET
END_PROPERTY

{attribute 'monitoring' := 'variable'}
PROPERTY DecelerationManual : LREAL
GET
DecelerationManual := lrDecelerationManual;
END_GET
SET
lrDecelerationManual := DecelerationManual;
END_SET
END_PROPERTY

METHOD Decouple : BOOL
VAR_INPUT
END_VAR
VAR
END_VAR
END_METHOD

METHOD PROTECTED Enable
VAR_INPUT
	bEnable		: BOOL;
END_VAR
// =========================================================

fbMCPower(	Enable 			:= bEnable, 
			Enable_Positive	:= bEnable, 
			Enable_Negative	:= bEnable, 
			Override		:= lrOverride,
			Axis			:= AxisRef,
			Status			=> bStatusEnable);
			
IF fbMcPower.Error THEN
	bError		:= TRUE;
	iErrorID 	:= fbMcPower.ErrorID;
END_IF

AxisRef.ReadStatus();
//bMoves := AxisRef.Status.Moving;

// =========================================================
END_METHOD

{attribute 'monitoring' := 'variable'}
PROPERTY Enabled : BOOL
GET
Enabled := bStatusEnable;
END_GET
END_PROPERTY

METHOD FirstCycle : BOOL
VAR_INPUT
	//ipAlarmController	:	I_AlarmController;
	//ipHMIController		:	I_HMIController;
	sName				:	STRING;
END_VAR
THIS^.sMotorName := sName;

//THIS^.ipAlarmController := ipAlarmController;
//ipAlarmController.AppendError(fbAxisError);

//THIS^.ipHMIController := ipHMIController;
//ipHMIController.AppendMotor(THIS^);
END_METHOD

{attribute 'monitoring' := 'variable'}
PROPERTY HaltDone : BOOL
GET
HaltDone := bHaltDone;
END_GET
END_PROPERTY

METHOD Home : BOOL // Start axis homing
VAR_INPUT
END_VAR
Home := FALSE;
END_METHOD

{attribute 'monitoring' := 'variable'}
PROPERTY Homed : BOOL
GET
Homed := AxisRef.Status.Homed;
END_GET
END_PROPERTY

{attribute 'monitoring' := 'variable'}
PROPERTY Homingable : BOOL
GET
Homingable := bHomingable;
END_GET
SET
bHomingable := Homingable;
END_SET
END_PROPERTY

METHOD Init : BOOL // Initialize axis
VAR_INPUT
END_VAR
IF iStepGeneral = 0 THEN
	iStepGeneral := 10;
END_IF

//Method output
	Init := (iStepGeneral >= 20);
END_METHOD

{attribute 'monitoring' := 'variable'}
PROPERTY Initialized : BOOL
GET
Initialized := bInitialized;
END_GET
END_PROPERTY

{attribute 'monitoring' := 'variable'}
PROPERTY JerkAuto : LREAL
GET
JerkAuto := lrJerkAuto;
END_GET
SET
lrJerkAuto := JerkAuto;
END_SET
END_PROPERTY

{attribute 'monitoring' := 'variable'}
PROPERTY JerkManual : LREAL
GET
JerkManual := lrJerkManual;
END_GET
SET
lrJerkManual := JerkManual;
END_SET
END_PROPERTY

METHOD Jog : BOOL // Do action 2 request, for instance: 'Pick and place unit' change tool (additional inputs needed)
VAR_INPUT
	Distance	:	LREAL;
END_VAR
IF iStepGeneral = 30 THEN
	iStepGeneral := 100;
END_IF

bMoveRelative := TRUE;
lrDistanceToGo := Distance;

//Method output
	Jog := (iStepGeneral = 110);
END_METHOD

{attribute 'monitoring' := 'variable'}
PROPERTY ManualMode : BOOL
GET
ManualMode := bManualMode;
END_GET
SET
bManualMode := ManualMode;
END_SET
END_PROPERTY

{attribute 'monitoring' := 'variable'}
PROPERTY MotorName : STRING
GET
MotorName := sMotorName;
END_GET
SET
sMotorName := MotorName;
END_SET
END_PROPERTY

METHOD MoveAbsolute : BOOL // Do action 2 request, for instance: 'Pick and place unit' change tool (additional inputs needed)
VAR_INPUT
	Position : LREAL;
END_VAR
IF (iStepGeneral = 30) OR ((iStepGeneral = 90) AND (Position<>lrPosition)) THEN
	iStepGeneral := 80;
END_IF

bMoveAbsolute := TRUE;
lrPosition := Position;

//Method output
	MoveAbsolute := (iStepGeneral = 90);
END_METHOD

METHOD MoveRelative : BOOL // Do action 2 request, for instance: 'Pick and place unit' change tool (additional inputs needed)
VAR_INPUT
	Distance	:	LREAL;
END_VAR
IF iStepGeneral = 30 THEN
	iStepGeneral := 100;
END_IF

bMoveRelative := TRUE;
lrDistanceToGo := Distance;

//Method output
	MoveRelative := (iStepGeneral = 110);
END_METHOD

METHOD MoveVelocity : BOOL // Move the axis with constant velocity velocity, the velocity can be changed during movement 
VAR_INPUT
	lrVelocityIn	:	LREAL;
END_VAR
IF iStepGeneral = 30 THEN
	iStepGeneral := 60;
END_IF

bMoveVelocity := TRUE;
lrVelocityAuto := lrVelocityIn;

//Method output
	MoveVelocity := fbMcMoveVelocity.InVelocity;//(iStepGeneral = 70);
END_METHOD

{attribute 'monitoring' := 'variable'}
PROPERTY Override : LREAL
GET
Override := lrOverride;
END_GET
SET
lrOverride := Override;
END_SET
END_PROPERTY

METHOD Reset : BOOL
VAR_INPUT
END_VAR
fbMcHalt(			Execute	:= FALSE,
					Axis 	:= AxisRef);
fbMcMoveVelocity(	Execute	:= FALSE,
					Axis 	:= AxisRef);
fbMcMoveAbsolute(	Execute	:= FALSE,
					Axis 	:= AxisRef);
fbMcMoveRelative(	Execute	:= FALSE,
					Axis 	:= AxisRef);
IF AxisRef.Status.Error THEN
	fbMcReset(		Execute	:= TRUE,
					Axis 	:= AxisRef);
ELSE
	fbMcReset(		Execute	:= FALSE,
					Axis 	:= AxisRef);
END_IF
bError := FALSE;
iErrorID := 0;
fbAxisError.Reset();
Reset := TRUE;
END_METHOD

{attribute 'monitoring' := 'variable'}
PROPERTY ResetDone : BOOL
GET
ResetDone := bResetDone;
END_GET
END_PROPERTY

METHOD PROTECTED StateAborting : BOOL
VAR_INPUT
END_VAR
bInitialized := FALSE;
CASE iStepAborting OF
	0: 	fbMcHalt(	Execute	:= FALSE,
					Axis 	:= AxisRef);
		fbMcMoveVelocity(	Execute	:= FALSE,
							Axis 	:= AxisRef);
		fbMcMoveAbsolute(	Execute	:= FALSE,
							Axis 	:= AxisRef);
		fbMcMoveRelative(	Execute	:= FALSE,
							Axis 	:= AxisRef);
		fbMcReset(			Execute	:= FALSE,
							Axis 	:= AxisRef);
		fbMcStop(			Execute	:= FALSE,
							Axis 	:= AxisRef);					
		iStepAborting := 10;
	10:	fbMcStop(	Execute	:= TRUE,
					Axis 	:= AxisRef,
					Jerk := lrJerkAuto,
					Deceleration := lrDecelerationAuto);
		IF fbMcStop.Done THEN
			iStepAborting := 20;
		ELSIF fbMcStop.Error THEN
			bError := fbMcStop.Error;
			iErrorID := fbMcStop.ErrorID;
			iStepAborting := 20;
		END_IF
	20:	fbMcStop(	Execute	:= FALSE,
					Axis 	:= AxisRef);
		iStepAborting := 0;
		iStepGeneral := 0;
							
END_CASE
END_METHOD

METHOD PROTECTED StateHalt
VAR_INPUT
	bDriveHalt		: BOOL;					// Request stop
END_VAR
//TODO: copied from sample, finish before use
// =========================================================

IF bDriveHalt THEN
	// Move Execute FALSE
	fbMcMoveVelocity(	Execute	:= FALSE,
				Axis 	:= AxisRef);
ELSE
	// Reset done signal
	bHaltDone := FALSE;
END_IF

// Trigger
fbTriggerHalt(CLK := bDriveHalt);

IF fbTriggerHalt.Q THEN
	fbMcHalt(	Execute	:= TRUE,
				Axis 	:= AxisRef);
ELSE
	fbMcHalt(Axis := AxisRef);
END_IF

// Done / Error / Command aborted
IF fbMcHalt.Done OR fbMcHalt.Error OR fbMcHalt.CommandAborted THEN
	bError		:= fbMcHalt.Error;
	iErrorID 	:= fbMcHalt.ErrorID;
	bHaltDone 	:= fbMcHalt.Done;
	
	fbMcMoveVelocity(	Execute	:= FALSE,
				Axis 	:= AxisRef);
				
	fbMcHalt(	Execute	:= FALSE,
				Axis 	:= AxisRef);
END_IF

// =========================================================
END_METHOD

METHOD PROTECTED StateInit : BOOL //Unit is performing initialization
VAR_INPUT
END_VAR
VAR
END_VAR
//Sequence
	CASE iStepInit OF
		0: 	// reset axis
				fbMcReset(	Axis := AxisRef,
							Execute := TRUE);
			IF 
				fbMcReset.Done
			THEN
				fbMcReset(	Axis := AxisRef,
							Execute := FALSE);
				iStepInit := 10;
			ELSIF
				fbMcReset.Error 
			THEN
				bError := TRUE;
				iErrorID := fbMcReset.ErrorID;	
			END_IF
			
		10: // axis ready
			IF
				AxisRef.Status.StandStill
			THEN
				iStepInit := 100;
			END_IF

		100: // initialized
			iStepGeneral := 20;
	END_CASE
END_METHOD

METHOD PROTECTED StateMachine : BOOL // Sate machien of unit
VAR_INPUT
END_VAR

VAR
	StateAction6Done: INT;
END_VAR
//State machine						   
	CASE iStepGeneral OF
		0:  //Uninitialized
			Enable(FALSE);
			StateUninitialized();
	
		10: //Initializing - reset, power on, 
			Enable(TRUE);
			StateInit();
	
		20: //Initialized-Ready - nothing to do
			Enable(TRUE);
			StateReady();
		
		30: //Ready to start - wait for action
			Enable(TRUE);
			StateReadyToStart();
	
(*		40: //homing
			Enable(TRUE);
			StateHoming();
			
		50: //Homing done
			Enable(TRUE);
			StateHomingDone();
*)			
		60: //move velocity
			Enable(TRUE);
			StateMovingVelocity();
			
		//70: //Move Velocity done

		80: //move ptp absolute
			Enable(TRUE);
			StateMovingAbsolute(lrPosition);

		90: //move ptp absolute done
			Enable(TRUE);
			StateMovingAbsoluteDone();			
		
		100: //move relative
			Enable(TRUE);
			StateMovingRelative(lrDistanceToGo);
			
		110: //move relative done
			Enable(TRUE);
			StateMovingRelativeDone();
					
		120: //stop
			Enable(TRUE);
			StateStopping();
			
		130: //stop done
			Enable(TRUE);
			StateStoppingDone();
			
		-10: //aborting
			Enable(TRUE);
			StateAborting();
	END_CASE
END_METHOD

METHOD PROTECTED StateMovingAbsolute : BOOL // Unit is performing action 2
VAR_INPUT
	Position:	LREAL;
END_VAR
VAR_INST


END_VAR
VAR
	lrVelocity		:	LREAL;
	lrAcceleration	:	LREAL;
	lrDeceleration	:	LREAL;
	lrJerk			:	LREAL;
END_VAR
// reinitialization of FB for different position
	IF (fbMcMoveAbsolute.Position<>Position) AND fbMcMoveAbsolute.Busy THEN
			fbMcMoveAbsolute(	Axis			:= AxisRef,
								Execute			:= FALSE,
								BufferMode		:= mcBufferMode);
			fbMcMoveAbsolute.FB_INIT(TRUE,TRUE);

			//RETURN;
	END_IF

// motion parameters
IF bManualMode THEN 
	lrVelocity 		:=	lrVelocityManual;
	lrAcceleration	:=	lrAccelerationManual;
	lrDeceleration	:=	lrDecelerationManual;
	lrJerk			:=	lrJerkManual;
ELSE
	lrVelocity 		:=	lrVelocityAuto;
	lrAcceleration	:=	lrAccelerationAuto;
	lrDeceleration	:=	lrDecelerationAuto;
	lrJerk			:=	lrJerkAuto;
END_IF

// execution 
IF NOT fbMcMoveAbsolute.Error THEN // no error behavior
	fbMcMoveAbsolute(	Axis			:= AxisRef,
						Execute			:= TRUE,
						Position		:= Position,
						Velocity		:= lrVelocity,
						Acceleration	:= lrAcceleration,
						Deceleration	:= lrDeceleration,
						Jerk			:= lrJerk,
						BufferMode		:= mcBufferMode);
						
	IF fbMcMoveAbsolute.Done AND AxisRef.Status.InTargetPosition THEN
		iStepGeneral := 90;
	END_IF
	
ELSE // error behavior
		bError		:= TRUE;
		iErrorID 	:= fbMcMoveAbsolute.ErrorID;
		fbMcMoveAbsolute(	Axis			:= AxisRef,
							Execute			:= FALSE);
END_IF
END_METHOD

METHOD PROTECTED StateMovingAbsoluteDone : BOOL // Unit is performing action 2
VAR_INPUT

END_VAR
VAR_INST

END_VAR
VAR
	lrVelocity		:	LREAL;
	lrAcceleration	:	LREAL;
	lrDeceleration	:	LREAL;
	lrJerk			:	LREAL;
END_VAR
fbMcMoveAbsolute(	Axis			:= AxisRef,
					Execute			:= FALSE);
IF NOT bMoveAbsolute THEN
		iStepGeneral := 30;
END_IF
END_METHOD

METHOD PROTECTED StateMovingRelative : BOOL // Unit is performing action 2
VAR_INPUT
	Distance	:	LREAL;
END_VAR

VAR
	lrVelocity		: LREAL;
	lrAcceleration	: LREAL;
	lrDeceleration	: LREAL;
	lrJerk			: LREAL;
END_VAR
// motion parameters
IF bManualMode THEN 
	lrVelocity := lrVelocityManual;
	lrAcceleration	:=	lrAccelerationManual;
	lrDeceleration	:=	lrDecelerationManual;
	lrJerk	:=	lrJerkManual;
ELSE
	lrVelocity := lrVelocityAuto;
	lrAcceleration	:=	lrAccelerationAuto;
	lrDeceleration	:=	lrDecelerationAuto;
	lrJerk	:=	lrJerkAuto;
END_IF

//Execute
IF NOT fbMcMoveRelative.Error THEN // no error behavior
	fbMcMoveRelative(	Axis			:= AxisRef,
						Execute			:= TRUE,
						Distance		:= Distance,
						Velocity		:= lrVelocity,
						Acceleration	:= lrAcceleration,
						Deceleration	:= lrDeceleration,
						Jerk			:= lrJerkAuto);
						
	IF fbMcMoveRelative.Done THEN
		iStepGeneral := 110;
	END_IF
ELSE // error behavior
	fbMcMoveRelative(	Axis			:= AxisRef,
						Execute			:= FALSE);
END_IF
END_METHOD

METHOD PROTECTED StateMovingRelativeDone : BOOL // Unit has finished action 2, waiting for release of the request
VAR_INPUT
END_VAR
fbMcMoveRelative(	Axis			:= AxisRef,
					Execute			:= FALSE);
					
IF NOT bMoveRelative THEN
	iStepGeneral := 30;
END_IF
END_METHOD

METHOD PROTECTED StateMovingVelocity : BOOL // Unit is performing action 2
VAR_INPUT
END_VAR
VAR_INST
	mcDirection	:MC_Direction;
	lrVelocityPreviousCycle :LREAL;
END_VAR
VAR
	FB_INIT: INT;
END_VAR
IF NOT fbMcMoveVelocity.Error THEN // no error behavior
	//	Instance management - new instance of MC_MoveVelocity called to dynamical change of motion parameters 
		IF VelocityAuto <> lrVelocityPreviousCycle THEN

			//fbMcMoveVelocity.FB_INIT(TRUE,TRUE);
			fbMcMoveVelocity(	Execute 		:= FALSE,
								Axis 			:= AxisRef);
		END_IF
	

	//direction choose
		IF VelocityAuto>=0 THEN
			mcDirection := MC_Positive_Direction;
		ELSE
			mcDirection := MC_Negative_Direction;
		END_IF
	
	// move
	IF VelocityAuto=0 THEN
		fbMcHalt(	Execute 		:= TRUE,
					Deceleration	:= DecelerationAuto,
					BufferMode		:= mcBufferMode,
					Axis 			:= AxisRef,
					Jerk	 		:= lrJerkAuto);
		fbMcMoveVelocity(	Execute 		:= FALSE,
							Velocity 		:= ABS(VelocityAuto),
							Acceleration	:= AccelerationAuto,
							Deceleration	:= DecelerationAuto,
							BufferMode		:= mcBufferMode,
							Direction 		:= mcDirection,
							Axis 			:= AxisRef,
							Jerk	 		:= lrJerkAuto);
	ELSE
		fbMcHalt(	Execute 		:= FALSE,
					Deceleration	:= DecelerationAuto,
					BufferMode		:= mcBufferMode,
					Axis 			:= AxisRef,
					Jerk	 		:= lrJerkAuto);
		fbMcMoveVelocity(	Execute 		:= TRUE,
							Velocity 		:= ABS(VelocityAuto),
							Acceleration	:= AccelerationAuto,
							Deceleration	:= DecelerationAuto,
							BufferMode		:= mcBufferMode,
							Direction 		:= mcDirection,
							Axis 			:= AxisRef,
							Jerk	 		:= lrJerkAuto);
	END_IF
		lrVelocityPreviousCycle := VelocityAuto;
ELSE // error behavior
	bError		:= TRUE;
	iErrorID 	:= fbMcMoveVelocity.ErrorID;
	fbMcMoveVelocity(	Execute	:= FALSE,
						Axis 	:= AxisRef);
END_IF
END_METHOD

METHOD PROTECTED StateReady : BOOL // Unit is initialized
VAR_INPUT
END_VAR
iStepGeneral := 30;
END_METHOD

METHOD PROTECTED StateReadyToStart : BOOL // Unit is ready to start the cycle/action, in this state some preparation that are not a part of initialization can be performed
VAR_INPUT
END_VAR
END_METHOD

METHOD PROTECTED StateStopping : BOOL // Unit is performing action 2
VAR_INPUT
END_VAR

VAR
	bDriveStop: BOOL;
	iGeneralStep: INT;
END_VAR
// Move Execute FALSE
	fbMcMoveVelocity(	Execute	:= FALSE,
						Axis 	:= AxisRef);
	fbMcMoveAbsolute(	Execute	:= FALSE,
						Axis 	:= AxisRef);
	fbMcMoveRelative(	Execute	:= FALSE,
						Axis 	:= AxisRef);
// stop axis
	fbMcStop(	Axis :=	AxisRef,
				Deceleration := DecelerationAuto,
				Jerk := JerkAuto,
				Execute := TRUE);
			
// Done / Error / Command aborted
IF fbMcStop.Error THEN
	bError		:= fbMcStop.Error;
	iErrorID 	:= fbMcStop.ErrorID;
	bHaltDone 	:= fbMcStop.Done;
				
	fbMcStop(	Execute	:= FALSE,
				Axis 	:= AxisRef);
ELSIF fbMcStop.Done THEN				
	iStepGeneral := 130;
	fbMcStop(	Execute	:= FALSE,
				Axis 	:= AxisRef);
END_IF
END_METHOD

METHOD StateStoppingDone : BOOL
VAR_INPUT
END_VAR
//do something if necessary
IF NOT bStop THEN
	iStepGeneral := 30;
END_IF
END_METHOD

METHOD PROTECTED StateUninitialized : BOOL // Unit is uninitialized
VAR_INST

END_VAR
bInitialized := FALSE;
END_METHOD

METHOD Stop : BOOL // Do action 2 request, for instance: 'Pick and place unit' change tool (additional inputs needed)
VAR_INPUT
END_VAR
IF iStepGeneral >= 30 AND iStepGeneral <> 130 THEN
	iStepGeneral := 120;
END_IF
bStop := TRUE;

//Method output
	Stop := (iStepGeneral = 130);
END_METHOD

{attribute 'monitoring' := 'variable'}
PROPERTY Unit : STRING
GET
Unit := sUnits;
END_GET
SET
sUnits:=Unit;
END_SET
END_PROPERTY

{attribute 'monitoring' := 'variable'}
PROPERTY VelocityAuto : LREAL
GET
VelocityAuto := lrVelocityAuto;
END_GET
SET
lrVelocityAuto := VelocityAuto;
END_SET
END_PROPERTY

{attribute 'monitoring' := 'variable'}
PROPERTY VelocityManual : LREAL
GET
VelocityManual := lrVelocityManual;
END_GET
SET
lrVelocityManual := VelocityManual;
END_SET
END_PROPERTY

END_FUNCTION_BLOCK

// ---- POUs/Alarm/FB_Alarm.TcPOU
FUNCTION_BLOCK FB_Alarm
VAR_INPUT
END_VAR
VAR_OUTPUT
END_VAR
VAR
	iAlarmNumber	:	UINT := 0;
	bTemporary		:	BOOL;
	bLatched		:	BOOL;
	sDescription	:	STRING;
	tsTimeOfOccur	:	TIMESTRUCT;
END_VAR

{attribute 'monitoring' := 'variable'}
PROPERTY AlarmNumber : UINT
GET
AlarmNumber := iAlarmNumber;
END_GET
SET
iAlarmNumber := AlarmNumber;
END_SET
END_PROPERTY

{attribute 'monitoring' := 'variable'}
PROPERTY Description : String
GET
Description := sDescription;
END_GET
SET
sDescription := Description;
END_SET
END_PROPERTY

METHOD Get : BOOL
VAR_INPUT
END_VAR
VAR_OUTPUT

END_VAR
Get := bLatched;
END_METHOD

METHOD Reset : BOOL
VAR_INPUT
END_VAR
IF NOT bTemporary THEN
	IF bLatched = TRUE THEN
		Reset := TRUE;
		bLatched := FALSE;
	END_IF
ELSE
	Reset := FALSE;
END_IF
END_METHOD

METHOD Set : BOOL
VAR
END_VAR
VAR_INPUT
	bIn	:	BOOL;
END_VAR
bTemporary := bIn;
IF NOT bLatched AND bIn THEN
	bLatched := TRUE;
	tsTimeOfOccur := GVL.fbLocalTime.systemTime;
END_IF
END_METHOD

PROPERTY TimeOfOccur : TIMESTRUCT
GET
TimeOfOccur := tsTimeOfOccur;
END_GET
END_PROPERTY

END_FUNCTION_BLOCK

// ---- POUs/UniversalBlocks/Cylinder/FB_CylinderDiag.TcPOU
(* FB_CylinderDiag	- number of control signals:
							one direction is controllable
					- type of feedback signal:
							feedback in base and work position
					- with position diagnosis						*)
					
FUNCTION_BLOCK FB_CylinderDiag EXTENDS FB_Cylinder
VAR_INPUT
	tTimeOut 	 		: TIME;			// Time for watchdog that monitores if cylinder reaches base/work position
END_VAR
VAR_OUTPUT
	bError				: BOOL;			// Error signal (diagnosed from position watchdog)
	sErrorMsg			: STRING;		// Error message
END_VAR
VAR
	fbTriggerError		: R_TRIG;		// Trigger to recognize rising edge of error
	bErrorMove			: BOOL;			// Move error
	fbTimerWatchDog		: TON;			// Watchdog timer for monitoring if cylinder reaches base/work position
END_VAR

// =========================================================
;
// =========================================================

METHOD PROTECTED Diag
VAR_INPUT
END_VAR
// =========================================================
// Timer starts when cylinder is not in base and work position
	
	IF NOT bAtBasePos AND NOT bAtWorkPos THEN
		fbTimerWatchDog(IN := TRUE,
						PT := tTimeOut);
	ELSE
		fbTimerWatchDog(IN := FALSE,
						PT := tTimeOut);
	END_IF

// =========================================================
// Error if cylinder does not reach base or work position
	
	fbTriggerError(CLK := fbTimerWatchDog.Q);
	
	bError := fbTimerWatchDog.Q;
	
	IF fbTriggerError.Q THEN
		bErrorMove := bMoveToWork;
	END_IF
	
	IF bError THEN
		IF bErrorMove = bMoveToWork THEN
			IF bMoveToWork THEN
				sErrorMsg := 'Work position not reached';
			ELSE
				sErrorMsg := 'Base position not reached';
			END_IF
		ELSE
			bError := FALSE;
			sErrorMsg := '';
		END_IF
	ELSE
		sErrorMsg := '';
	END_IF

// =========================================================
END_METHOD

METHOD Reset
VAR_INPUT
END_VAR
// =========================================================

// Calling method Reset of base class FB_Cylinder via 'SUPER^.'
SUPER^.Reset();		

// Reset error
bError 		:= FALSE;
sErrorMsg 	:= '';

// =========================================================
END_METHOD

METHOD PROTECTED StateMachine
VAR_INPUT
	bBasePosReq		: BOOL;
	bWorkPosReq		: BOOL;
END_VAR
// =========================================================

IF NOT bError THEN
	// Calling method StateMachine of base class FB_Cylinder via 'SUPER^.'
	SUPER^.StateMachine(bBasePosReq := bBasePosReq,
						bWorkPosReq	:= bWorkPosReq );
	
	// Diagnosis
	Diag();
END_IF

// =========================================================
END_METHOD

END_FUNCTION_BLOCK

// ---- POUs/UniversalBlocks/Cylinder/FB_Cylinder.TcPOU
(* FB_Cylinder		- number of control signals:
							one direction is controllable
					- type of feedback signal:
							feedback in base and work position		*)
						
FUNCTION_BLOCK FB_Cylinder
VAR_INPUT
	bAtBasePos		AT %I*	: BOOL;		// Hardware input signal: cylinder is at base position
	bAtWorkPos		AT %I*	: BOOL;		// Hardware input signal: cylinder is at work position
END_VAR
VAR_OUTPUT
	bMoveToWork		AT %Q*	: BOOL;		// Hardware output signal to move cylinder to work position
	bMoveToBase		AT %Q*	: BOOL;		// Hardware output signal to move cylinder to base position
END_VAR

// =========================================================
;
// =========================================================

PROPERTY PUBLIC bState_AtBasePos : BOOL
GET
bState_AtBasePos := bAtBasePos;
END_GET
END_PROPERTY

PROPERTY PUBLIC bState_AtWorkPos : BOOL
GET
bState_AtWorkPos := bAtWorkPos;
END_GET
END_PROPERTY

PROPERTY bState_MoveToBase : bool
GET
bState_MoveToBase := bMoveToBase;
END_GET
END_PROPERTY

PROPERTY PUBLIC bState_MoveToWork : BOOL
GET
bState_MoveToWork := bMoveToWork;
END_GET
END_PROPERTY

METHOD MoveToBase
VAR_INPUT
END_VAR
// =========================================================
	
StateMachine(	bBasePosReq := TRUE,
				bWorkPosReq	:= FALSE );
							
// =========================================================
END_METHOD

METHOD MoveToWork
VAR_INPUT
END_VAR
// =========================================================
	
StateMachine(	bBasePosReq := FALSE,
				bWorkPosReq	:= TRUE );
								
// =========================================================
END_METHOD

METHOD Reset
VAR_INPUT
END_VAR
// =========================================================

bMoveToWork := FALSE;
bMoveToBase	:= TRUE;

// =========================================================
END_METHOD

METHOD PROTECTED StateMachine
VAR_INPUT
	bBasePosReq		: BOOL;
	bWorkPosReq		: BOOL;
END_VAR
// =========================================================
// Base or work position requested
		
	IF bWorkPosReq THEN
		bMoveToWork := TRUE;
		bMoveToBase	:= FALSE;
	END_IF
	
	IF bBasePosReq THEN
		bMoveToWork := FALSE;
		bMoveToBase	:= TRUE;
	END_IF

// =========================================================
END_METHOD

END_FUNCTION_BLOCK

// ---- POUs/UniversalBlocks/Cylinder/FB_CylinderTemp.TcPOU
(* FB_CylinderTemp	- number of control signals:
							one direction is controllable
					- type of feedback signal:
							feedback in base and work position
					- with temperature signal					*)

FUNCTION_BLOCK FB_CylinderTemp EXTENDS FB_Cylinder
VAR_INPUT
	fTempCurrent	AT %I*	: LREAL;		// Hardware input signal: cylinder temperature
END_VAR

// =========================================================
;
// =========================================================

END_FUNCTION_BLOCK

// ---- POUs/UniversalBlocks/Cylinder/FB_CylinderTempDiag.TcPOU
(* FB_CylinderTempDiag		- number of control signals:
									one direction is controllable
							- type of feedback signal:
									feedback in base and work position
							- with temperature diagnosis					*)

FUNCTION_BLOCK FB_CylinderTempDiag EXTENDS FB_CylinderTemp
VAR_INPUT
	fTempMax		AT %I*	: LREAL;		// Global input signal: maximal allowed cylinder temperature for temperature monitoring
	fTempMin		AT %I*	: LREAL;		// Global input signal: minimal allowed cylinder temperature for temperature monitoring
END_VAR
VAR_OUTPUT
	bError					: BOOL;			// Error signal (diagnosed from temperature monitoring)
	sErrorMsg				: STRING;		// Error message
END_VAR

// =========================================================
;
// =========================================================

METHOD PROTECTED Diag
VAR_INPUT
END_VAR
// =========================================================
// Error if temperatur of cylinder is not in accepted interval
	
	bError := NOT (fTempCurrent >= fTempMin AND fTempCurrent <= fTempMax);
	
	IF bError THEN
		IF fTempCurrent > fTempMax THEN
			sErrorMsg := 'Temperature above maximum';
		ELSE
			sErrorMsg := 'Temperature below minimum';
		END_IF
	ELSE
		sErrorMsg := '';
	END_IF

// =========================================================
END_METHOD

METHOD Reset
VAR_INPUT
END_VAR
// =========================================================
	
// Calling method Reset of base class FB_Cylinder via 'SUPER^.'
SUPER^.Reset();			

// Reset error
bError 		:= FALSE;
sErrorMsg 	:= '';

// =========================================================
END_METHOD

METHOD PROTECTED StateMachine
VAR_INPUT
	bBasePosReq		: BOOL;
	bWorkPosReq		: BOOL;
END_VAR
// =========================================================

IF NOT bError THEN
	// Calling method StateMachine of base class FB_Cylinder via 'SUPER^.'
	SUPER^.StateMachine(bBasePosReq := bBasePosReq,
						bWorkPosReq	:= bWorkPosReq );
	
	// Diagnosis
	Diag();
END_IF

// =========================================================
END_METHOD

END_FUNCTION_BLOCK

// ---- POUs/UniversalBlocks/Cylinder/FB_CylinderTempRecord.TcPOU
(* FB_CylinderTempRecord	- number of control signals:
									one direction is controllable
							- type of feedback signal:
									feedback in base and work position
							- with temperature recording for data analysis		*)

FUNCTION_BLOCK FB_CylinderTempRecord EXTENDS FB_CylinderTemp
VAR_INPUT
	bRecordStart		: BOOL;						// Signal to start the temperature recording
	tIntervalTime		: TIME;						// Time of intervals to record the temperature 
END_VAR
VAR_OUTPUT
	bRecordDone			: BOOL;						// True if the temperature recording is done
	aTemps				: ARRAY[1..100] OF LREAL;	// Array with recorded temperatures
END_VAR
VAR
	fbTimerInterval		: TON;						// Timer to control the recording interval
	nIndex				: INT;						// Index to handle temperature array
END_VAR

// =========================================================
;
// =========================================================

METHOD Record
VAR_INPUT
END_VAR
// =========================================================
// Recording array filled
	
	bRecordDone := (nIndex = 100);

// =========================================================
// Recording temperatures
	
	IF bRecordStart AND NOT bRecordDone AND NOT fbTimerInterval.Q THEN
		fbTimerInterval(IN := TRUE,
						PT := tIntervalTime );
	END_IF
	
	IF fbTimerInterval.Q THEN
		fbTimerInterval(IN := FALSE);
		
		nIndex 			:= nIndex + 1;
		aTemps[nIndex] 	:= fTempCurrent;
	END_IF

// =========================================================
END_METHOD

METHOD Reset
VAR_INPUT
END_VAR
// =========================================================

// Calling method Reset of base class FB_Cylinder via 'SUPER^.'
SUPER^.Reset();

// Reset temperature array
FOR nIndex := 1 TO 100 BY 1 DO
	aTemps[nIndex] := 0;
END_FOR

// Reset index
nIndex := 0;

// =========================================================
END_METHOD

END_FUNCTION_BLOCK

// ---- POUs/UniversalBlocks/Universal motor/FB_Axis_Multi_Master.TcPOU
FUNCTION_BLOCK FB_Axis_Multi_Master EXTENDS FB_Axis
VAR
		// =============== Axis reference =========================
	Master1AxisRef			: AXIS_REF;	
	Master2AxisRef			: AXIS_REF;	
	Master3AxisRef			: AXIS_REF;	
	Master4AxisRef			: AXIS_REF;	
	
	// =============== Motion function blocks =================
	fbGearInMultiMaster: MC_GearInMultiMaster; //FB to gear in multiple axes
	fbGearOut: MC_GearOut; //FB to gear out multiple axes
	
	lrGearRatio1	:	LREAL;
	lrGearRatio2	:	LREAL;
	lrGearRatio3	:	LREAL;
	lrGearRatio4	:	LREAL;
	
END_VAR

SUPER^();

METHOD Abort : BOOL
VAR_INPUT
END_VAR
SUPER^.Abort();
END_METHOD

METHOD Couple : BOOL
VAR_INPUT

END_VAR

VAR

END_VAR
IF iStepGeneral = 30 THEN
	iStepGeneral := 1000;
END_IF

Couple := iStepGeneral = 1010;
END_METHOD

METHOD Decouple : BOOL
VAR_INPUT

END_VAR

VAR
	bGearInMultimaster	:	BOOL;
END_VAR
IF iStepGeneral = 1010 OR iStepGeneral = 1000 THEN
	iStepGeneral := 1020;
END_IF
Decouple := iStepGeneral = 30;
END_METHOD


PROPERTY GearRatio1 : LREAL
GET
GearRatio1 := lrGearRatio1;
END_GET
SET
lrGearRatio1 := GearRatio1;
END_SET
END_PROPERTY


PROPERTY GearRatio2 : LREAL
GET
GearRatio2 := lrGearRatio2;
END_GET
SET
lrGearRatio2 := GearRatio2;
END_SET
END_PROPERTY


PROPERTY GearRatio3 : LREAL
GET
GearRatio3 := lrGearRatio3;
END_GET
SET
lrGearRatio3 := GearRatio3;
END_SET
END_PROPERTY


PROPERTY GearRatio4 : LREAL
GET
GearRatio4 := lrGearRatio4;
END_GET
SET
lrGearRatio4 := GearRatio4;
END_SET
END_PROPERTY

METHOD Reset : BOOL
VAR_INPUT
END_VAR
fbGearInMultiMaster(	Slave 			:= AxisRef,
						Enable 			:= FALSE,
						Master1			:= Master1AxisRef,
						Master2			:= Master2AxisRef,
						Master3			:= Master3AxisRef,
						Master4			:= Master4AxisRef,);
fbGearOut(	Slave	:= AxisRef,
			Execute	:= FALSE);
						
SUPER^.Reset();
END_METHOD

METHOD PROTECTED StateAborting : BOOL
VAR_INPUT
END_VAR
VAR
END_VAR
CASE iStepAborting OF
	0: 	fbMcHalt(	Execute	:= FALSE,
					Axis 	:= AxisRef);
		fbMcMoveVelocity(	Execute	:= FALSE,
							Axis 	:= AxisRef);
		fbMcMoveAbsolute(	Execute	:= FALSE,
							Axis 	:= AxisRef);
		fbMcMoveRelative(	Execute	:= FALSE,
							Axis 	:= AxisRef);
		fbMcReset(			Execute	:= FALSE,
							Axis 	:= AxisRef);
		fbGearInMultiMaster(	Enable			:= FALSE,
								Master1			:= Master1AxisRef,
								Master2			:= Master2AxisRef,
								Master3			:= Master3AxisRef,
								Master4			:= Master4AxisRef,
								Slave			:= AxisRef);
		fbGearOut (		Execute	:= FALSE,
						Slave 	:= AxisRef);
		fbMcStop(		Execute	:= FALSE,
						Axis 	:= AxisRef);
		iStepAborting := 10;
	10: fbGearOut(	Execute := TRUE,
					Slave := AxisRef);
		IF fbGearOut.Done THEN
			iStepAborting := 15;
		ELSIF fbGearOut.Error THEN
			bError := TRUE;
			iErrorID := fbGearOut.ErrorID;
			iStepAborting := 15;
		END_IF
	15: fbGearOut(	Execute := FALSE,
					Slave := AxisRef);
		iStepAborting := 20;
		
	20:	fbMcStop(	Execute	:= TRUE,
					Axis 	:= AxisRef);
		IF fbMcStop.Done THEN
			iStepAborting := 30;
		ELSIF fbMcStop.Error THEN
			bError := fbMcStop.Error;
			iErrorID := fbMcStop.ErrorID;
			iStepAborting := 30;
		END_IF
	30:	fbMcStop(	Execute	:= FALSE,
					Axis 	:= AxisRef);
		iStepAborting := 0;
		iStepGeneral := 0;
							
END_CASE
END_METHOD

METHOD PROTECTED StateCoupleDone : BOOL
VAR_INPUT
END_VAR
fbGearInMultiMaster(	Enable			:= TRUE,
						Master1			:= Master1AxisRef,
						GearRatio1		:= lrGearRatio1,
						Master2			:= Master2AxisRef,
						GearRatio2		:= lrGearRatio2,
						Master3			:= Master3AxisRef,
						GearRatio3		:= lrGearRatio3,
						Master4			:= Master4AxisRef,
						GearRatio4		:= lrGearRatio4,
						Slave			:= AxisRef,
						Acceleration	:= lrAccelerationAuto);
END_METHOD

METHOD PROTECTED StateCoupling : BOOL
VAR_INPUT
END_VAR
fbGearInMultiMaster(	Enable			:= TRUE,
						Master1			:= Master1AxisRef,
						GearRatio1		:= lrGearRatio1,
						Master2			:= Master2AxisRef,
						GearRatio2		:= lrGearRatio2,
						Master3			:= Master3AxisRef,
						GearRatio3		:= lrGearRatio3,
						Master4			:= Master4AxisRef,
						GearRatio4		:= lrGearRatio4,
						Slave			:= AxisRef,
						Acceleration	:= lrAccelerationAuto);
IF fbGearInMultiMaster.InGear THEN
	iStepGeneral := 1010;
END_IF
END_METHOD

METHOD PROTECTED StateDecoupling : BOOL
VAR_INPUT
END_VAR
fbGearInMultiMaster(	Enable			:= FALSE,
						Master1			:= Master1AxisRef,
						GearRatio1		:= lrGearRatio1,
						Master2			:= Master2AxisRef,
						GearRatio2		:= lrGearRatio2,
						Master3			:= Master3AxisRef,
						GearRatio3		:= lrGearRatio3,
						Master4			:= Master4AxisRef,
						GearRatio4		:= lrGearRatio4,
						Slave			:= AxisRef,
						Acceleration	:= lrAccelerationAuto);
fbGearOut(	Slave := AxisRef,
			Execute := TRUE);
			
IF fbGearOut.Done THEN
	fbGearOut(	Slave := AxisRef,
				Execute := FALSE);
	iStepGeneral := 30;
END_IF
END_METHOD

METHOD PROTECTED StateMachine : BOOL // Sate machien of unit
VAR_INPUT
END_VAR

VAR
	StateAction6Done: INT;
END_VAR
//State machine	
SUPER^.StateMachine();					   
	CASE iStepGeneral OF
		1000:  // Gearing in MM
			Enable(TRUE);
			StateCoupling();
	
		1010: // Gearing in MM done 
			Enable(TRUE);
			StateCoupleDone();
	
		1020: // Gearing out MM
			Enable(TRUE);
			StateDecoupling();
	END_CASE
END_METHOD

END_FUNCTION_BLOCK

// ---- POUs/UniversalBlocks/Universal motor/FB_HomeableAxis.TcPOU
FUNCTION_BLOCK FB_HomeableAxis EXTENDS FB_Axis
VAR_INPUT
END_VAR
VAR_OUTPUT
END_VAR
VAR
	fbMcHome		: MC_Home;				// FB to home axis
	bDoHoming		:	BOOL; //do action 1 variable
	piHomeSensor	: FB_Input;
END_VAR

(*
	- Version: V2.0
	- Modified: SOHN
	- Time: 20/10/2021
	- Description: Change bHomeSensor into FB_Input: piHomeSensor so that fbHMI can append input. Modify Stop() 
	- Comment: May the moral be with you!!
*)

	IF bFirstCycle THEN
		piHomeSensor.Description := 'Home Detector';
	END_IF

	bHomingable := TRUE;
	bDoHoming := FALSE;
	Super^();

METHOD Home : BOOL // Start axis homing
VAR_INPUT
END_VAR
IF iStepGeneral = 30 THEN
	iStepGeneral := 40;
END_IF

bDoHoming := TRUE;

//Method output
	Home := (iStepGeneral = 50);
END_METHOD

PROPERTY HomeDetector : I_Input
GET
HomeDetector := piHomeSensor;
END_GET
END_PROPERTY

METHOD Reset : BOOL
VAR_INPUT
END_VAR
fbMcHome(			Execute	:= FALSE,
					Axis 	:= AxisRef);
SUPER^.Reset();
END_METHOD

METHOD PROTECTED StateAborting : BOOL
VAR_INPUT
END_VAR
bInitialized := FALSE;
CASE iStepAborting OF
	0: 
		fbMcHome(			Execute	:= FALSE,
							Axis 	:= AxisRef);
END_CASE
Super^.StateAborting();
END_METHOD

METHOD PROTECTED StateHoming : BOOL // Unit is performing action 1
VAR_INPUT
END_VAR
IF NOT fbMcHome.Error THEN // no error behavior

//Home
	fbMcHome(		Execute 	:= TRUE,
					Axis		:= AxisRef,
					HomingMode	:= MC_DefaultHoming,
					bCalibratioNCam		:= piHomeSensor.Value);
	IF fbMcHome.Done THEN
		iStepGeneral := 50;
		fbMcHome(	Execute 	:= FALSE,
					Axis		:= AxisRef,
					HomingMode	:= MC_DefaultHoming,
					bCalibratioNCam		:= piHomeSensor.Value);
	END_IF

ELSE // error behavior
	fbMcHome(		Execute 	:= FALSE,
					Axis		:= AxisRef,
					HomingMode	:= MC_DefaultHoming,
					bCalibratioNCam		:= piHomeSensor.Value);
					
	bError		:= TRUE;
	iErrorID 	:= fbMcHome.ErrorID;
END_IF
END_METHOD

METHOD PROTECTED StateHomingDone : BOOL // Unit has finished action 1, waiting for release of the request
VAR_INPUT
END_VAR
//do something if necessary
IF NOT bDoHoming THEN
	iStepGeneral := 30;
END_IF
END_METHOD

METHOD PROTECTED StateMachine : BOOL // Sate machien of unit
VAR_INPUT
END_VAR

VAR
	StateAction6Done: INT;
END_VAR
//State machine						   
	CASE iStepGeneral OF
		40: //homing
			Enable(TRUE);
			StateHoming();
			
		50: //Homing done
			Enable(TRUE);
			StateHomingDone();
	END_CASE
	
Super^.StateMachine();
END_METHOD

END_FUNCTION_BLOCK

// ---- POUs/UniversalBlocks/Universal motor/FB_HomeableEncAxis.TcPOU
FUNCTION_BLOCK FB_HomeableEncAxis EXTENDS FB_HomeableAxis
VAR_INPUT
END_VAR
VAR_OUTPUT
END_VAR
VAR
	fbEncWait : TON;
	bEnableLatchC AT %Q*: BOOL;
END_VAR

	IF bFirstCycle THEN
		piHomeSensor.Description := 'Encoder C track';
	END_IF

	SUPER^();

METHOD PROTECTED StateHoming : BOOL // Unit is performing action 1
VAR_INPUT
END_VAR
IF NOT fbMcHome.Error THEN // no error behavior

//Home
	fbMcHome(		Execute 	:= TRUE,
					Axis		:= AxisRef,
					HomingMode	:= MC_DefaultHoming,
					bCalibratioNCam		:= piHomeSensor.Value);
	
	bEnableLatchC := TRUE;
	fbEncWait(IN := piHomeSensor.Value, PT:= T#1000MS);
	bEnableLatchC R= fbEncWait.Q;
	
	IF fbMcHome.Done THEN
		iStepGeneral := 50;
		fbMcHome(	Execute 	:= FALSE,
					Axis		:= AxisRef,
					HomingMode	:= MC_DefaultHoming,
					bCalibratioNCam		:= piHomeSensor.Value);
		bEnableLatchC := FALSE;
	END_IF

ELSE // error behavior
	fbMcHome(		Execute 	:= FALSE,
					Axis		:= AxisRef,
					HomingMode	:= MC_DefaultHoming,
					bCalibratioNCam		:= piHomeSensor.Value);
	
	bEnableLatchC := FALSE;
	bError		:= TRUE;
	iErrorID 	:= fbMcHome.ErrorID;
END_IF
END_METHOD

END_FUNCTION_BLOCK
